TYPE st_csv :
STRUCT
	dia: STRING;
	mes: STRING;
	ano: STRING;
	ordem: STRING;
	lote: string;
END_STRUCT
END_TYPE

(* stored: Version 1.1.0.1, ProductVersion 3.1.4024.12
   DUT st_csv: Id {639e3da9-11ee-4691-a7b1-93f5cc203242} *)
